TYPE Read_ISPS_Values_To_PC_Struct :
UNION
	S_ISPSValues_To_PC:S_ISPSValues_To_PC_Struct;
END_UNION
END_TYPE

(* stored: Version 1.1.0.1, ProductVersion 3.1.4024.16
   DUT Read_ISPS_Values_To_PC_Struct: Id {a78aed47-db45-4aac-bd69-5dd9493d594b} *)
